(* CoDeSys 2.3.9.50 project: flat-BC9000.pr6 *)
(* Libraries: PlcHelperBC.lb6 7.5.01 11:03:00, COMlibV2.lb6 25.2.14 08:37:08, ModbusRTU.lb6 13.5.15 12:37:26, standard.lb6 5.6.98 11:03:02 *)

(* Global variable list: Globale_Variablen *)
VAR_GLOBAL

	Clear						: ClearComBuffer;
	TxBufferCom1				: ComBuffer;
	RxBufferCom1				: ComBuffer;
	SerialLineControlCom1			: SerialLineControl;
	ReceiveDataCom1			: ReceiveData;
	SendDataCom1				: SendData;

	Modbus						: Modbus_Struct;
	Internal						: Internal_Struct;

	HW_vent_out_level					AT	%QW2:WORD:=7000;(* Напряжение управления вытяжным вентилятором (0-32767) *)
(*	HW_vent_out_level2					AT	%QW6:WORD:=7000;
	HW_vent_out_level3					AT	%QW10:WORD:=7000;
	HW_vent_out_level4					AT	%QW14:WORD:=7000;
*)

(*	RS485read.MB.InData AT %IB16 : MB_KL6inData22B;
	RS485read.MB.OutData AT %QB16 : MB_KL6outData22B;
*)


	HW_temp_kitchen_box					AT %IW42:INT; (*Температура на кухне в коробе  *)
	HW_temp_vent_in						AT %IW46:INT; (*Температура притока перед фильтром *)
	HW_temp_street						AT %IW50:INT; (*Температура на улице *)
	HW_temp_bedroom					AT %IW54:INT; (*Температура в спальне *)

	HW_temp_child_small_room			AT %IW58:INT; (*Температура *)
	HW_temp_kitchen						AT %IW62:INT; (*Температура *)
	HW_temp_child_big_room				AT %IW66:INT; (*Температура *)


	HW_vent_in_trans_105_130				AT	%QX72.0:BOOL:=FALSE;  (* Напряжение 110 или 130 В *)
	HW_vent_in_trans_160_220				AT	%QX72.1:BOOL:=TRUE;  (* Напряжение 160 или 220 В *)
	HW_vent_in_trans_LO_HI				AT	%QX72.2:BOOL:=FALSE;  (* Напряжение 110/130  или 160/220 В *)
	HW_steam							AT	%QX72.3:BOOL:=FALSE; (* Разрешение включения увлажнителя *)

	HW_vent_out							AT	%QX72.4:BOOL:=FALSE; (* Вытяжной вентилятор*)
	HW_kitchen_vent_out					AT	%QX72.5:BOOL:=FALSE; (*Надплитная вытяжка*)
	HW_vent_in_heat_level				AT	%QX72.6:BOOL:=FALSE; (* Подогрев притока ночной режим   -5 К ТЭН *)
	HW_vent_valve						AT	%QX72.7:BOOL:=FALSE; (*Клапан приточной вентиляции"*)


	HW_valve_water_kitchen				AT	%QX73.0:BOOL; (* Кран ХВС и ГВС на кухне *)
	HW_valve_water_bathroom				AT	%QX73.1:BOOL; (* Кран ХВС и ГВС в санузле *)
	HW_LIGHT_ALL						AT	%QX73.2:BOOL; (*Свет в квартире *)
	HW_LIGHT_hall						AT	%QX73.3:BOOL; (*Ночной/аварийный свет в коридоре *)

(*
	HW_rez1								AT	%QX69.4:BOOL; 
	HW_rez2								AT	%QX69.5:BOOL; 
	HW_rez3								AT	%QX69.6:BOOL; 
	HW_rez4								AT	%QX69.7:BOOL;

*)

	HW_trans_power						AT	%QX74.0:BOOL:=FALSE; (*Подача тока на трансформатор и реле ТЭН-а *)
	HW_vent_in_heat						AT	%QX74.1:BOOL:=FALSE; (* Подогрев притока - ТЭН *)





	HW_sensor_fld_kitchen				AT %IX72.0:BOOL; (* Датчик протечки на кухне*)
	HW_sensor_fld_tlt						AT %IX72.1:BOOL; (* Датчик протечки в туалете*)
	HW_sensor_fld_post					AT %IX72.2:BOOL; (* Датчик протечки в постирочной*)
	HW_sensor_fld_van					AT %IX72.3:BOOL; (* Датчик протечки в ванной*)
	HW_impulse_kitchen_water_cold		AT %IX72.4:BOOL; (* Счётчик холодной воды на кухне*)
	HW_impulse_kitchen_water_warm		AT %IX72.5:BOOL; (* Счётчик горячей воды на кухне*)
	HW_vent_reay_pressure				AT %IX72.6:BOOL; (*Реле давления*)
	HW_kitchen_button_vent_out			AT %IX72.7:BOOL; (* Кнопка кухонной вытяжки*)

	HW_sensor_vent_valve_closed			AT %IX73.0:BOOL;
	HW_sensor_vent_valve_opened		AT %IX73.1:BOOL;
	HW_IN01							AT %IX73.2:BOOL;(*Кнопка вкл и откл света в квартире*)
	HW_IN02							AT %IX73.3:BOOL;(*Кнопка вкл и откл кранов воды на кухне*)
	HW_IN03							AT %IX73.4:BOOL;(*Кнопка вкл и откл кранов воды на кухне*)
	HW_IN04							AT %IX73.5:BOOL;(*Кнопка вкл и откл Вентиляции*)
	HW_IN05							AT %IX73.6:BOOL;(*Кнопка вкл и откл Резерв*)
	HW_gerkon							AT %IX73.7:BOOL;(*Датчик открытия двери - геркон*)


	HW_PIR_door						AT %IX74.0:BOOL;(*Датчик открытия двери - pir *)
	HW_PIR_hall							AT %IX74.1:BOOL;(*Датчик открытия двери - pir *)
	HW_electro							AT %IX74.2:BOOL;(*Датчик наличия электроэнергии*)
	HW_battery_low						AT %IX74.3:BOOL;(*Датчик низкого напряжения  АКБ*)



	HW_impulse_bathroom_water_cold		AT %IX75.0:BOOL; (* Счётчик горячей воды санузла NAMUR*)
	HW_impulse_bathroom_water_warm		AT %IX75.2:BOOL; (* Счётчик холодной воды санузла NAMUR*)







END_VAR

(* Global variable list: Variable_Configuration *)
VAR_CONFIG
	RS485read.MB.InData AT %IB16 : MB_KL6inData22B;
	RS485read.MB.OutData AT %QB16 : MB_KL6outData22B;
END_VAR

(* Data type *)
TYPE Internal_struct :
STRUCT

	Temp_vent_in						:	REAL; 		(*16434*)
	City_hum 							:	REAL;		(*16436*)
	Kitchen_room_tempout					:	REAL;		(*16438 *)

	Kitchen_room_temp 					:	REAL; 		(*16440 *)
	Kitchen_room_temp_SHT20 			:	REAL;		(*16442 *)
	Kitchen_room_hum 					:	REAL;		(*16444 *)
	Kitchen_room_CO2					:	REAL;		(*16446  *)

	Child_small_room_temp 				:	REAL; 		(* 16448 *)
	Child_small_room_temp_SHT20 		:	REAL;	(*16450 *)
	Child_small_room_hum 				:	REAL;	(*16452 *)
	Child_small_room_CO2 				:	REAL;	(* 16454 *)

	Child_big_room_temp	 				:	REAL; 	(* 16456 *)
	Child_big_room_temp_SHT20	 		:	REAL;	(* 16458 *)
	Child_big_room_hum	 				:	REAL;	(* 16460 *)
	Child_big_room_CO2	 				:	REAL;	(* 16462 *)

	Bed_room_temp	 					:	REAL; 	(* 16464 *)
	Bed_room_temp_SHT20				:	REAL;	(* 16466 *)
	Bed_room_hum	 					:	REAL;	(* 16468 *)
	Bed_room_CO2						:	REAL;	(*16470 *)

END_STRUCT
END_TYPE

(* Data type *)
TYPE Modbus_struct :
STRUCT

	(* MEED TO SAVE IN MEMORY*)



	Vent							AT %MB0	:	BOOL;	(*16384*)
	Vent_out						AT %MB2	:	BOOL;	(*16385*)
	Vent_heat					AT %MB4	:	INT;		(*16386*)
	Vent_heat_level				AT %MB6	:	BOOL;	(*16387*)
	Vent_valve_status				AT %MB8	:	INT;     	(*16388*)
	Steam						AT %MB10	:	BOOL;	(*16389*)
	Target_CO2					AT %MB12	:	INT;		(*16390*)
	Target_hum					AT %MB14	:	INT; 	(*16391*)
	Security_status				AT %MB16	:	BOOL;	(*16392*)
(*	Light_reserv					AT %MB18	:	BOOL;*)   (*16393*)
	Light						AT %MB20	:	BOOL; 	(*16394 *)
	Light_hall					AT %MB22	:	BOOL; 	(*16395*)

	Kitchen_stat_cold_water		AT %MD24	:	DINT; (* 16396*)
	Kitchen_stat_warm_water		AT %MD28	:	DINT; (* 16398*)
	Bathroom_stat_cold_water		AT %MD32	:	DINT; (* 16400*)
	Bathroom_stat_warm_water		AT %MD36	:	DINT; (* 16402*)

	FLD_valve_kitchen 			AT %MB40	:	BOOL; (* Положение  крана воды на кухне 16404*)
	FLD_valve_bathroom 			AT %MB42	:	BOOL; (*Положение  крана воды в санузле 16405*)
	FLD_ALRM_KITCHEN 			AT %MB44	:	BOOL; (*ТРЕВОГА ЗАТОПЛЕНИЕ НА КУХНЕ 16406*)
	FLD_ALRM_BATH 			AT %MB46	:	BOOL; (*ТРЕВОГА ЗАТОПЛЕНИЕ В САНУЗЛЕ 16407*)

	(* NOT NEED TO SAVE in MEMORY *)

	Steam_level						AT %MB48	:	INT;     (* 16408*)
	Steam_status						AT %MB50	:	INT;  (* 16409*)
	Steam_real						AT %MB52	:	INT; (* 16410*)
	Vent_input_level					AT %MB54	:	INT;		(*16411*)
	Vent_output_level					AT %MB56	:	INT; 	(*0-100%    16412 *)
	Vent_pressure_relay				AT %MB58	:	BOOL; (* 16413*)


	Gerkon							AT %MB60	:	BOOL; (*Датчик открытия входной двери (геркон)    16414 *)
	PIR_door						AT %MB62	:	BOOL;(*Датчик открытия входной двери PIR-штора   16415 *)
	Power_supply					AT %MB64	:	BOOL;(*Электроэнергия   16416 *)
	Battery_low						AT %MB66	:	BOOL;	(* 16417*)
	Rezerv							AT %MB68	:	BOOL; (* 16418*)

	FLD_PRC						AT %MB70	:	BOOL; (*Датчик в постирочной 16419*)
	FLD_TLT						AT %MB72	:	BOOL; (*Датчик в туалете 16420*)
	FLD_BATH						AT %MB74	:	BOOL;(*Датчик в  ванной 16421*)
	FLD_KUH						AT %MB76	:	BOOL;(*Датчик на  кухне 16422*)

	Uv								AT %MW80	:	DINT;		(*16424*)
	Ia								AT %MW84	:	DINT;		(*16426*)
	Pw								AT %MW88	:	DINT;		(*16428*)
	E_T1							AT %MW92	:	DINT;		(*16430*)
	E_T2							AT %MW96	:	DINT;		(*16432*)


	Temp_vent_in					AT %MW100	:	DINT; 		(*16434*)
	City_hum 						AT %MW104	:	DINT;		(*16436*)
	Kitchen_room_tempout				AT %MW108	:	DINT;		(*16438 *)

	Kitchen_room_temp 				AT %MW112	:	DINT; 		(*16440 *)
	Kitchen_room_temp_SHT20 		AT %MW116	:	DINT;		(*16442 *)
	Kitchen_room_hum 				AT %MW120	:	DINT;		(*16444 *)
	Kitchen_room_CO2				AT %MW124	:	DINT;		(*16446  *)

	Child_small_room_temp 			AT %MW128	:	DINT; 		(* 16448 *)
	Child_small_room_temp_SHT20 	AT %MW132	:	DINT;	(*16450 *)
	Child_small_room_hum 			AT %MW136	:	DINT;	(*16452 *)
	Child_small_room_CO2 			AT %MW140	:	DINT;	(* 16454 *)

	Child_big_room_temp	 			AT %MW144	:	DINT; 	(* 16456 *)
	Child_big_room_temp_SHT20	 	AT %MW148	:	DINT;	(* 16458 *)
	Child_big_room_hum	 			AT %MW152	:	DINT;	(* 16460 *)
	Child_big_room_CO2	 			AT %MW156	:	DINT;	(* 16462 *)

	Bed_room_temp	 				AT %MW160	:	DINT; 	(* 16464 *)
	Bed_room_temp_SHT20			AT %MW164	:	DINT;	(* 16466 *)
	Bed_room_hum	 				AT %MW168	:	DINT;	(* 16468 *)
	Bed_room_CO2					AT %MW172	:	DINT;	(*16470 *)





END_STRUCT
END_TYPE

(* POU MAIN, ST *)
PROGRAM MAIN
VAR
	SW_LIGHT				: SM_BUTT;		(* вкл/откл  света в квартире *)
	SW_VALVE_BATH		: SM_BUTT;
	SW_VALVE_KITCHEN		: SM_BUTT;
	SW_VENT				: SM_BUTT_SHORT_LONG;		(* вкл/откл вентиляции *)
	SW_REZERV			: SM_BUTT_TIMER;

END_VAR
	RS485read;				(* Работа с устройствами на шине RS485 *)
	Ventcontrol;				(* Глобальный контроль вентустановки*)
	VentPower;				(* Авторегулировка мощности вентустановки по датчикам CO2*)
	Counters;				(* Счётчики воды *)
	Fluid_bath;				(* Защита от протечки в санузлах. Оработка нажатия физической и виртульной кнопки №2 *)
	Fluid_kitchen;				(* Защита от протечки в кухне. Оработка нажатия физической и виртульной кнопки №3 *)
	Light_hall;				(* Свет в коридоре *)




(* Оработка нажатия физических и виртульных кнопок №1, №4, №5 *)

	SW_LIGHT 				(IN:=HW_IN01, IN1:= Modbus.Light, 	Q=>NOT Modbus.Light);	(* Конпка №1 *)
	SW_VALVE_BATH 		(IN:=HW_IN02, IN1:= Modbus.FLD_valve_bathroom, 	Q=>NOT Modbus.FLD_valve_bathroom);	(* Конпка №2 *)
	SW_VALVE_KITCHEN 	(IN:=HW_IN03, IN1:= Modbus.FLD_valve_kitchen,	Q=>NOT Modbus.FLD_valve_kitchen);	(* Конпка №3 *)
	SW_VENT 				(bIn:=HW_IN04, TC:=t#2000ms);		(* Конпка №4  , обработка короткого и долгого нажатия *)
	SW_REZERV		 	(IN:=HW_IN05,Q=>);	(* Конпка №3 *)

	IF	SW_VENT.bSingle	THEN
		Modbus.Vent	:= NOT Modbus.Vent;
	END_IF

	IF	SW_VENT.bLong	THEN
		Modbus.Steam	:= NOT Modbus.Steam;
	END_IF

(* Прямая связь между экспортирумымми переменными и  переменными, жестко привязаными  к физ. портам. Частота обновления= циклу ПЛК  : *)

	HW_LIGHT_ALL				:=	NOT Modbus.Light;				(* СВЕТ в квартире*)
	HW_LIGHT_HALL				:=	Modbus.Light_hall;					(* Аварийный СВЕТ в квартире*)
	Modbus.Gerkon				:=	HW_gerkon;						(* Геркон на двери*)
	Modbus.PIR_door				:=	HW_pir_door;						(* Датчик движения на двери *)
	Modbus.Power_supply			:=	HW_electro;						(* Датчик наличия электроэнергии *)
	Modbus.Battery_low			:=	HW_battery_low;					(* Датчик наличия электроэнергии *)
	Modbus.Vent_pressure_relay	:=	HW_vent_reay_pressure; 	(* Relay pressure *)
	HW_vent_in_heat_level		:=	Modbus.Vent_heat_level;

	Internal.Temp_vent_in				:=	INT_TO_REAL(HW_temp_vent_in)/10;
	Internal.Kitchen_room_tempout		:=	INT_TO_REAL(HW_temp_street)/10;
	Internal.Bed_room_temp			:=	INT_TO_REAL(HW_temp_bedroom)/10;
	Internal.Kitchen_room_temp			:=	INT_TO_REAL(HW_temp_kitchen)/10;
	Internal.Child_big_room_temp		:=	INT_TO_REAL(HW_temp_child_big_room)/10;
	Internal.Child_small_room_temp		:=	INT_TO_REAL(HW_temp_child_small_room)/10;



	Modbus.Temp_vent_in				:=	INT_TO_DINT(HW_temp_vent_in);
	Modbus.Kitchen_room_tempout		:=	INT_TO_DINT(HW_temp_street);
	Modbus.Bed_room_temp			:=	INT_TO_DINT(HW_temp_bedroom);
	Modbus.Kitchen_room_temp		:=	INT_TO_DINT(HW_temp_kitchen);
	Modbus.Child_big_room_temp		:=	INT_TO_DINT(HW_temp_child_big_room);
	Modbus.Child_small_room_temp	:=	INT_TO_DINT(HW_temp_child_small_room);


IF (Modbus.Security_status = FALSE AND HW_electro = FALSE  ) THEN
	Modbus.Light_hall :=TRUE;
END_IF

IF (Modbus.Security_status = TRUE ) THEN
	Modbus.Light_hall := FALSE;
END_IF
END_PROGRAM

(* POU SM_BUTT, ST *)
FUNCTION_BLOCK SM_BUTT            (* ФУНКЦИОНАЛЬНЫЙ БЛОК ДЛЯ ПРОСТОЙ КНОПКИ *)
    VAR_INPUT
       	IN: BOOL;          	(*ВХОД ЗА КОТОРЫМ МЫ СЛЕДИМ *)
	IN1:BOOL;				(*ВЫХОД ЗА КОТОРЫМ ТОЖЕ СЛЕДИМ*)
    END_VAR

    VAR_OUTPUT
	Q : BOOL;        			(*СОСТОЯНИЕ ВЫХОДА*)
    END_VAR
    VAR
  MEM : BOOL;    			(* ВНУТРЕННЯЯ ПЕРЕМЕННАЯ ДЛЯ ХРАНЕНИЯ СОСТОЯНИЯ КНОПКИ *)
    END_VAR
Q:=IN1;

IF IN AND NOT MEM THEN 	(* ПОЙМАЛИ ПЕРЕДНИЙ ФРОНТ - НАЖАЛИ НА КНОПКУ *)
	Q := NOT IN1;    			(* МЕНЯЕМ СОСТОЯНИЕ ВЫХОДА НА ПРОТИВОПОЛОЖНОЕ *)
END_IF

MEM := IN;                       		(* ЗАПОМИНАЕМ ТЕКУЩЕЕ ЗНАЧЕНИЕ КНОПКИ *)
END_FUNCTION_BLOCK

(* POU SM_BUTT_SHORT_LONG, ST *)
FUNCTION_BLOCK SM_BUTT_SHORT_LONG
VAR_INPUT
	bIn 	: BOOL;
	TC	: TIME := t#2000ms;
END_VAR
VAR_OUTPUT
	bSingle	: BOOL;
	bLong 	: BOOL;
END_VAR
VAR
	timer 	: TP;
	ft1		: F_TRIG;
	ft2		: F_TRIG;
END_VAR
timer(in := bIn, pt := TC);

ft1(clk := bIn);
bSingle := ft1.Q AND timer.Q;

ft2(clk := timer.Q);
bLong := ft2.Q AND bIn;
END_FUNCTION_BLOCK

(* POU SM_BUTT_TIMER, ST *)
FUNCTION_BLOCK SM_BUTT_TIMER            (* ФУНКЦИОНАЛЬНЫЙ БЛОК ДЛЯ ПРОСТОЙ КНОПКИ *)
    VAR_INPUT
       	IN: BOOL;          	(*ВХОД ЗА КОТОРЫМ МЫ СЛЕДИМ *)
    END_VAR

    VAR_OUTPUT
	Q : BOOL;        			(*СОСТОЯНИЕ ВЫХОДА*)
    END_VAR

VAR
	RT1				: R_TRIG;
	tmCheck			: TON;
END_VAR
tmCheck;

RT1(clk := IN);

IF RT1.Q THEN
	Modbus.Rezerv	:=	TRUE;
	tmCheck(in:=FALSE);
	tmCheck(in:=TRUE,pt:=t#2s);
END_IF

IF tmCheck.Q	THEN
		Modbus.Rezerv	:=	FALSE;
END_IF
END_FUNCTION_BLOCK

(* POU RS485read, ST *)
PROGRAM RS485read
VAR
	MB: ModbusRtuMaster_KL6x22B;
	timeoutvalue					: TIME := T#500ms;		(* timeout while waiting for an answer of the modbus slave *)
	delta_sensor_hum				: INT:=10;					(*Корректировка показаний датчика, % относительной влажности*)
	Period_steam				: INT := 60; 				(* Частота изменения уставки мощности  увлажнителя, секунды*)
	Period_modbus				: INT := 10;  				(* Частота опроса устройств modbus, секунды*)

	r_Target_hum					: REAL;
	r_room_hum					: REAL;
	i_Steam_level				: INT:=0;
	MBdata						: ARRAY [1..2] OF INT;		(* The size of this array can be adapted to the modbus slaves register area *)

	sensors_SHT20_v1_id			: ARRAY[1..4] OF BYTE:=16#01, 16#02, 16#03, 16#37;
	sensors_SHT20_v1_hum		: ARRAY[1..4] OF REAL:=4(0);
	sensors_SHT20_v1_temp		: ARRAY[1..4] OF REAL:=4(0);


	sensors_CO2_id				: ARRAY[1..4] OF BYTE:=16#68, 16#65, 16#66, 16#67;
	sensors_CO2_ppm			: ARRAY[1..4] OF REAL;

	FtrigBusy					: F_TRIG;
	state						: INT;
	busy						: BOOL;
	LastErrorstate					: INT;
	LastModbusError				: ST_ModbusErrorDiagnostics;
	CounterError					: DINT;
	CounterSuccess				: DINT;
	tmCheck						: TON;
	Timer1						: TON;
	Timer2						: TON;
	Timer1Q						: BOOL;
	Timer2Q						: BOOL;
	Hum_old						: REAL;
	Steam_response				: WORD:=0;
	tTimerValue					: TIME;
	tTimerValue_modbus			: TIME;
	get_run_Merc200_done		: BOOL;
	get_hist_Merc200_done		: BOOL;
	get_run_Merc200				: FB_GET_RUN_MERC200;
	get_hist_Merc200				: FB_GET_HIST_MERC200;


	i: INT:=1;
	k: INT:=1;

END_VAR
tmcheck();
Timer1();
Timer2();

CASE state OF

0:
		MB.ReadRegs(Execute:= FALSE);
		state := 2;


 2:
	Clear(Buffer := RxBufferCom1);


		MB.ReadRegs(
			UnitID:= sensors_SHT20_v1_id[i],
			Quantity:= 2,
			MBAddr:= 0,
			cbLength:= 6,
			pMemoryAddr:= ADR(MBdata),
			Execute:= TRUE,
			Timeout:= timeoutvalue,
			Busy => busy,
		);
		IF NOT busy THEN
			IF (mb.Error = FALSE ) THEN
				sensors_SHT20_v1_temp[i]:=INT_TO_REAL(MBdata[1]);
				sensors_SHT20_v1_hum[i]:=INT_TO_REAL(MBdata[2])- 10*delta_sensor_hum;
			END_IF
			i:=i+1;
			MB.ReadRegs(Execute:= FALSE);
			IF (i>4 )	THEN
				i:=1;

				Internal.Kitchen_room_hum				:=	sensors_SHT20_v1_hum[1];
				Internal.Bed_room_hum				:=	sensors_SHT20_v1_hum[2];
				Internal.Child_big_room_hum			:=	sensors_SHT20_v1_hum[3];
				Internal.Child_small_room_hum			:=	sensors_SHT20_v1_hum[4];

(*				Internal.Kitchen_room_temp_SHT20		:=	sensors_SHT20_v1_temp[1];
				Internal.Bed_room_temp_SHT20			:=	sensors_SHT20_v1_temp[2];
				Internal.Child_small_room_temp_SHT20	:=	sensors_SHT20_v1_temp[4];
				Internal.Child_big_room_temp_SHT20	:=	sensors_SHT20_v1_temp[3];

				Modbus.Kitchen_room_temp_SHT20		:=	REAL_TO_INT(sensors_SHT20_v1_temp[1]);
				Modbus.Bed_room_temp_SHT20		:=	REAL_TO_INT(sensors_SHT20_v1_temp[2]);
				Modbus.Child_big_room_temp_SHT20	:=	REAL_TO_INT(sensors_SHT20_v1_temp[3]);
				Modbus.Child_small_room_temp_SHT20	:=	REAL_TO_INT(sensors_SHT20_v1_temp[4]);
*)
				Modbus.Kitchen_room_hum				:=	REAL_TO_INT(sensors_SHT20_v1_hum[1]);
				Modbus.Bed_room_hum				:=	REAL_TO_INT(sensors_SHT20_v1_hum[2]);
				Modbus.Child_big_room_hum			:=	REAL_TO_INT(sensors_SHT20_v1_hum[3]);
				Modbus.Child_small_room_hum			:=	REAL_TO_INT(sensors_SHT20_v1_hum[4]);
				state :=26;
			ELSE
				state :=2;
			END_IF

		END_IF


26:
		MB.ReadInputRegs(
			UnitID:=sensors_CO2_id[k], (* station address *)
			Quantity:= 1,
			MBAddr:= 3,
			cbLength:= 4,
			pMemoryAddr:= ADR(MBdata),
			Execute:= TRUE,
			Timeout:= timeoutvalue,
			Busy => busy	);
		IF NOT busy THEN
			IF (mb.Error = FALSE ) THEN
				sensors_CO2_ppm[k]	:=	INT_TO_REAL(MBdata[1]);
			END_IF
			k:=k+1;
			MB.ReadRegs(Execute:= FALSE);
			IF (k>4 )	THEN
				k:=1;
				Internal.Kitchen_room_CO2		:=	sensors_CO2_ppm[1];
				Internal.Bed_room_CO2		:=	sensors_CO2_ppm[2];
				Internal.Child_big_room_CO2	:=	sensors_CO2_ppm[3];
				Internal.Child_small_room_CO2	:=	sensors_CO2_ppm[4];

				Modbus.Kitchen_room_CO2		:=	REAL_TO_DINT(sensors_CO2_ppm[1]);
				Modbus.Bed_room_CO2		:=	REAL_TO_DINT(sensors_CO2_ppm[2]);
				Modbus.Child_big_room_CO2	:=	REAL_TO_DINT(sensors_CO2_ppm[3]);
				Modbus.Child_small_room_CO2	:=	REAL_TO_DINT(sensors_CO2_ppm[4]);

				state :=47;
			ELSE
				state :=26;
			END_IF
		END_IF

47:	(*Изменение уставки мощности увлажнителя при необходимости с частотой Period_steam *)

		IF (Modbus.Steam=TRUE AND Modbus.Vent=TRUE ) THEN
			r_Target_hum:=INT_TO_REAL( Modbus.Target_Hum) ;
			r_room_hum:=DINT_TO_REAL(Modbus.Bed_room_hum)/10;
			tTimerValue := t#60s;
			Timer2(IN:=NOT Timer2Q , PT:=tTimerValue , Q=>Timer2Q , ET=> );
			IF timer2.q THEN
				IF  ( r_room_hum <= r_Target_hum*0.5 AND i_Steam_level< 50 ) THEN
					i_Steam_level:=50;
				END_IF

				IF ( ( r_room_hum <=   Hum_old )
				AND ( r_room_hum > r_Target_hum*0.5)
				AND ( r_room_hum < r_Target_hum*0.95 )) THEN
					i_Steam_level:=i_Steam_level+1;
				END_IF

				IF ( r_room_hum >= r_Target_hum*1.05) THEN
					i_Steam_level:=i_Steam_level-1;
				END_IF

				Hum_old:=r_room_hum;

			END_IF

			IF (i_Steam_level>100) THEN
				i_Steam_level:=100;
			END_IF

			IF (i_Steam_level<10) THEN
				i_Steam_level:=10;
			END_IF

			Modbus.Steam_level:=INT_TO_BYTE(i_Steam_level);

			MB.WriteSingleRegister(
					UnitID:= 16#0A, (* station address *)
					Quantity:= 1,
					MBAddr:= 1537,
					cbLength:= 2,
					pMemoryAddr:= ADR(Modbus.Steam_level),
					Execute:= TRUE,
					Timeout:= timeoutvalue,
					Busy => busy	);
			IF NOT busy THEN
					MB.WriteSingleRegister(Execute:= FALSE);
					state := 77;
			END_IF
		ELSE
			Modbus.Steam_level:=0;
			state := 77;
		END_IF


77:		(* Фактический процент текущей  мощности увлажнителя *)

			MB.ReadRegs(
					UnitID:= 16#0A, (* station address *)
					Quantity:= 1,
					MBAddr:= 261,
					cbLength:= 2,
					pMemoryAddr:= ADR(Steam_response),
					Execute:= TRUE,
					Timeout:= timeoutvalue,
					Busy => busy	);
				IF NOT busy THEN
					IF (mb.Error = FALSE ) THEN
						Modbus.Steam_real:=Steam_response;
					END_IF
					MB.ReadRegs(Execute:= FALSE);
					state := 79;

				END_IF


79:
		tmCheck(in:=FALSE);
		tmCheck(in:=TRUE,pt:=t#2s);
		get_run_Merc200_done := FALSE;
		busy:=TRUE;
		get_run_Merc200( Uv=>Modbus.Uv,Ia=>Modbus.Ia,Pw=>Modbus.Pw, done=>get_run_Merc200_done);
		IF get_run_Merc200_done = TRUE THEN

			busy:=FALSE;
			state:=80;
		ELSIF tmcheck.Q THEN
			busy:=FALSE;
			 state:=80;
		END_IF

80:
		tmCheck(in:=FALSE);
		tmCheck(in:=TRUE,pt:=t#2s);
		get_hist_Merc200_done := FALSE;
		busy:=TRUE;
		get_hist_Merc200( E_T1=>Modbus.E_T1,E_T2=>Modbus.E_T2, done=>get_hist_Merc200_done);
		IF get_hist_Merc200_done = TRUE THEN

			busy:=FALSE;
			state:=88;
		ELSIF tmcheck.Q THEN
			busy:=FALSE;
			 state:=88;
		END_IF

88:
		tTimerValue_modbus := t#10s;
		Timer1(IN:=NOT Timer1Q , PT:=tTimerValue_modbus , Q=>Timer1Q , ET=> );
		IF timer1.q THEN

			state:=0;
		END_IF

END_CASE

FtrigBusy(CLK:=mb.BUSY );
IF FtrigBusy.Q THEN
	IF mb.Error THEN
		LastModbusError := mb.ErrorDiagnostics;
		LastErrorstate := state;
		CounterError := CounterError + 1;
	ELSE
		CounterSuccess := CounterSuccess + 1;
	END_IF
END_IF

SerialLinecontrolCom1(
	mode:=SerialLinemode_kl6_22b_standard,
	pComIn:=ADR(RS485read.MB.InData),
	pComOut:=ADR(RS485read.MB.OutData),
	SizeComIn:=SIZEOF(RS485read.MB.OutData),
	TxBuffer:=TxBufferCom1,
	RxBuffer:=RxBufferCom1,
	Error=>,
	errorid=>);
END_PROGRAM

(* POU FB_GET_RUN_MERC200, ST *)
FUNCTION_BLOCK FB_GET_RUN_MERC200
VAR_INPUT

END_VAR

VAR_OUTPUT
	Uv				: DINT;
	Ia				: DINT;
	Pw				: DINT;
	done			: BOOL;
END_VAR

VAR
	SendBuffer		: ARRAY[1..7] OF BYTE;
	ReceiveBuffer	: ARRAY[1..14] OF BYTE;
	Clear			: ClearComBuffer;
	state			: INT:= 0;
	tmcheck			: TON;

	crctest			: WORD;
	Uv_word			: WORD;
	Ia_word			: WORD;
	Pw_dword		: DWORD;

	CRC_calc: WORD;
	CRC_get: WORD := 1;

END_VAR
tmcheck();

CASE state OF

0:
	done:=FALSE;
	Clear(Buffer := RxBufferCom1);
	SendBuffer[1] := 16#00;

	SendBuffer[2] := 16#0B; (* Address  dec 740964 = hex 0B 4E 64  *)
	SendBuffer[3] := 16#4E; (* Address *)
	SendBuffer[4] := 16#64; (* Address *)

	SendBuffer[5] := 16#63; (*Command*)
	crctest:=F_CRC16(ADR(SendBuffer), 5);
	MEMCPY(ADR(SendBuffer)+5,ADR(crctest),2);

	SendDataCom1(pSendData:=ADR(SendBuffer),length:=7,TXbuffer:=TXBufferCom1,Busy=>,Error=>);

	tmCheck(in:=FALSE);
	tmCheck(in:=TRUE,pt:=t#2s);
	state:=1;

1: (*ответ*)

	ReceiveDataCom1(pPrefix:=,LenPrefix:=,pSuffix:=,LenSuffix:=,pReceiveData:=ADR(ReceiveBuffer),SizeReceiveData:=14,TImeOut:=t#2s,Reset:=,RXbuffer:=RxBufferCom1,DataReceived=>,busy=>,RxTimeout=>,LenReceiveData=>);

	IF ReceiveDataCom1.Error <> 0 THEN
		state:=9;
	END_IF

	IF ReceiveDataCom1.DataReceived THEN
		state:=2;
	ELSIF tmcheck.Q THEN
		 state:=9;
	END_IF;



2:(*расшифровка*)
	CRC_calc := F_CRC16(ADR(ReceiveBuffer), 12);
	MEMCPY(ADR(CRC_get),ADR(ReceiveBuffer[13]),1);
	MEMCPY(ADR(CRC_get)+1,ADR(ReceiveBuffer[14]),1);


	IF (  ReceiveBuffer[1] = 16#00  AND CRC_calc = CRC_get ) THEN

		MEMCPY(ADR(Uv_word),ADR(ReceiveBuffer[7]),1);
		MEMCPY(ADR(Uv_word)+1,ADR(ReceiveBuffer[6]),1);
		Uv:=STRING_TO_DINT(DWORD_TO_STRH(Uv_word));



		MEMCPY(ADR(Ia_word),ADR(ReceiveBuffer[9]),1);
		MEMCPY(ADR(Ia_word)+1,ADR(ReceiveBuffer[8]),1);
		Ia:=STRING_TO_DINT(DWORD_TO_STRH(Ia_word));

		MEMCPY(ADR(Pw_dword),ADR(ReceiveBuffer[12]),1);
		MEMCPY(ADR(Pw_dword)+1,ADR(ReceiveBuffer[11]),1);
		MEMCPY(ADR(Pw_dword)+2,ADR(ReceiveBuffer[10]),1);
		Pw:=STRING_TO_DINT(DWORD_TO_STRH(Pw_dword));


		state:=10;
	ELSE
		state:=9;
	END_IF

9:
	Uv:=0;
	done := TRUE;
	state:=0;
10:
	done := TRUE;
	state:=0;

END_CASE;
END_FUNCTION_BLOCK

(* POU MB_func/F_CRC16, ST *)
FUNCTION F_CRC16 : WORD
VAR_INPUT
	pData: POINTER TO BYTE;		(* указатель на блок данных *)
	Size: WORD;						(* размер блока  данных *)
END_VAR
VAR
	Cnt: BYTE;							(* счетчик битов *)
END_VAR
F_CRC16 := 16#FFFF;
WHILE Size > 0 DO
	F_CRC16 := F_CRC16 XOR pData^;
	FOR Cnt := 0 TO 7 DO
		IF F_CRC16.0 = 0 THEN
			F_CRC16 := SHR(F_CRC16, 1);
		ELSE
			F_CRC16 := SHR(F_CRC16, 1) XOR 16#A001;
		END_IF
	END_FOR;
	pData := pData + 1;
	Size := Size - 1;
END_WHILE
END_FUNCTION

(* POU DWORD_TO_STRH, ST *)
FUNCTION DWORD_TO_STRH : STRING(8)
VAR_INPUT
	IN : DWORD;
END_VAR
VAR
	i : INT;
	temp : BYTE;
	pt : POINTER TO BYTE;
END_VAR
(*
version 1.3	29. mar. 2008
programmer 	hugo
tested by	tobias

DWORD_TO_STRINGH converts a DWORD to a String of Hexadecimal represented by '0' .. '9' and 'A' .. 'F'.
The lowest order Character will be on the right and the high order Character on the left.

*)

(* @END_DECLARATION := '0' *)
(* read output adress to pointer *)
pt := ADR(DWORD_TO_STRH) + 8;
(* wirte the closing byte for the string *)
pt^:= 0;

(* write the 8 hex characters backwards *)
FOR i := 1 TO 8 DO;
	(* decrement the pointer *)
	pt := pt - 1;
	(* read the lowest order hex value *)
	temp := DWORD_TO_BYTE(in AND 16#0000000F);
	(* convert value to hex character *)
	IF temp <= 9 THEN temp := temp + 48; ELSE temp := temp + 55; END_IF;
	(* write character to output string *)
	PT^ := temp;
	(* shift in for nect hex character *)
	in := SHR(in,4);
END_FOR;


(* code beofre rev 1.2
FOR i := 1 TO 8 DO
	X := DWORD_TO_BYTE(in AND 2#1111);
	IF X <= 9 THEN X := X + 48; ELSE X := X + 55; END_IF;
	Cx := CHR(X);
	temp := CONCAT(Cx, temp);
	in := SHR(in,4);
END_FOR;
DWORD_TO_STRH := temp;
*)


(* revision history
hm	9. jun. 2007	rev 1.0		
	original version 

hm	11. sep. 2007	rev 1.1
	changed coding for compatibility with twincat, concat cannot support a function as an argument.

hm	15. dec. 2007	rev 1.2
	changed code for better performance

hm	29. mar. 2008	rev 1.3
	changed STRING to STRING(8)

*)
END_FUNCTION

(* POU FB_GET_HIST_MERC200, ST *)
FUNCTION_BLOCK FB_GET_HIST_MERC200
VAR_INPUT

END_VAR

VAR_OUTPUT
	E_T1			: DINT;
	E_T2			: DINT;
(*	E_T3			: REAL;
	E_T4			: REAL;
*)
	done			: BOOL;
END_VAR

VAR
	SendBuffer		: ARRAY[1..7] OF BYTE;
	ReceiveBuffer	: ARRAY[1..23] OF BYTE:=0,0,0,0,0,0,0,0,0,0,0,0,0,0,0,0,0,0,0,0,0,0,0;
	Clear			: ClearComBuffer;
	state			: INT:= 0;
	tmcheck			: TON;

	crctest			: WORD;
	T1_dword		: DWORD;
	T2_dword		: DWORD;
(*	T3_dword		: DWORD;
	T4_dword		: DWORD;
*)
	CRC_calc: WORD;
	CRC_get: WORD := 1;

END_VAR
tmcheck();

CASE state OF

0:
	done:=FALSE;
	Clear(Buffer := RxBufferCom1);
	SendBuffer[1] := 16#00;

	SendBuffer[2] := 16#0B; (* Address  dec 740964 =0B 4E 64    *)
	SendBuffer[3] := 16#4E; (* Address *)
	SendBuffer[4] := 16#64; (* Address *)

	SendBuffer[5] := 16#27; (*Command*)

	crctest:=F_CRC16(ADR(SendBuffer), 5);
	MEMCPY(ADR(SendBuffer)+5,ADR(crctest),2);

	SendDataCom1(pSendData:=ADR(SendBuffer),length:=7,TXbuffer:=TXBufferCom1,Busy=>,Error=>);

	tmCheck(in:=FALSE);
	tmCheck(in:=TRUE,pt:=t#2s);
	state:=1;

1: (*ответ*)

	ReceiveDataCom1(pPrefix:=,LenPrefix:=,pSuffix:=,LenSuffix:=,pReceiveData:=ADR(ReceiveBuffer),SizeReceiveData:=23,TImeOut:=t#2s,Reset:=,RXbuffer:=RxBufferCom1,DataReceived=>,busy=>,RxTimeout=>,LenReceiveData=>);

	IF ReceiveDataCom1.Error <> 0 THEN
		state:=9;
	END_IF

	IF ReceiveDataCom1.DataReceived THEN
		state:=2;
	ELSIF tmcheck.Q THEN
		 state:=9;
	END_IF;



2:(*расшифровка*)
	CRC_calc := F_CRC16(ADR(ReceiveBuffer), 21);
	MEMCPY(ADR(CRC_get),ADR(ReceiveBuffer[22]),1);
	MEMCPY(ADR(CRC_get)+1,ADR(ReceiveBuffer[23]),1);


	IF (  ReceiveBuffer[1] = 16#00  AND ReceiveBuffer[2] = 16#0B AND ReceiveBuffer[3] = 16#4E AND ReceiveBuffer[4] = 16#64  AND ReceiveBuffer[5] = 16#27) THEN

		MEMCPY(ADR(T1_dword),ADR(ReceiveBuffer[9]),1);
		MEMCPY(ADR(T1_dword)+1,ADR(ReceiveBuffer[8]),1);
		MEMCPY(ADR(T1_dword)+2,ADR(ReceiveBuffer[7]),1);
		MEMCPY(ADR(T1_dword)+3,ADR(ReceiveBuffer[6]),1);
		E_T1:=STRING_TO_DINT(DWORD_TO_STRH(T1_dword));
(*		E_T1:=DWORD_TO_DINT(T1_dword); *)

		MEMCPY(ADR(T2_dword),ADR(ReceiveBuffer[13]),1);
		MEMCPY(ADR(T2_dword)+1,ADR(ReceiveBuffer[12]),1);
		MEMCPY(ADR(T2_dword)+2,ADR(ReceiveBuffer[11]),1);
		MEMCPY(ADR(T2_dword)+3,ADR(ReceiveBuffer[10]),1);
		E_T2:=STRING_TO_DINT(DWORD_TO_STRH(T2_dword));
(*		E_T2:=DWORD_TO_DINT(T2_dword); *)
(*
		MEMCPY(ADR(T3_dword),ADR(ReceiveBuffer[17]),1);
		MEMCPY(ADR(T3_dword)+1,ADR(ReceiveBuffer[16]),1);
		MEMCPY(ADR(T3_dword)+2,ADR(ReceiveBuffer[15]),1);
		MEMCPY(ADR(T3_dword)+3,ADR(ReceiveBuffer[14]),1);
		E_T3:=0.01*STRING_TO_REAL(DWORD_TO_HEXSTR(T3_dword,1,FALSE));

		MEMCPY(ADR(T4_dword),ADR(ReceiveBuffer[21]),1);
		MEMCPY(ADR(T4_dword)+1,ADR(ReceiveBuffer[20]),1);
		MEMCPY(ADR(T4_dword)+2,ADR(ReceiveBuffer[19]),1);
		MEMCPY(ADR(T4_dword)+3,ADR(ReceiveBuffer[18]),1);
		E_T4:=0.01*STRING_TO_REAL(DWORD_TO_HEXSTR(T4_dword,1,FALSE));
*)
		state:=10;
	ELSE
		state:=9;
	END_IF

9:
	E_T1:=0;
	E_T2:=0;

	done := TRUE;
	state:=0;
10:
	done := TRUE;
	state:=0;

END_CASE;
END_FUNCTION_BLOCK

(* POU Ventcontrol, ST *)
PROGRAM VentControl
VAR
	Temperature_max_to_heat		: REAL:=17;		(* Максимальная температура наружнего воздуха при которой разрешено включать воздухонагреватель *)
	Temperature_min_for_steam	: REAL:=14;		(* Минимальная температура воздуха в вент канале для разрешения работы увлажнителя *)
	gisterezis					: REAL:=0.2;		(* Гистерезис  разрешения включения воздухонагревателя, градусы цельсия *)


END_VAR
(* Состояние приточного клапана *)

IF (HW_sensor_vent_valve_opened=TRUE) THEN
	Modbus.Vent_valve_status:=1;
END_IF

IF (HW_sensor_vent_valve_closed=TRUE) THEN
	Modbus.Vent_valve_status:=0;
END_IF

IF (HW_sensor_vent_valve_closed=FALSE AND HW_sensor_vent_valve_opened=FALSE) THEN
	Modbus.Vent_valve_status:=2;
END_IF


IF (HW_kitchen_button_vent_out=TRUE) THEN	(* Если активирована кнопка надплитной вытяжки*)
	HW_vent_out:=TRUE;						(* Включаем вытяжной вент *)
	HW_vent_out_level:=32767;					(* Подаём управляющий сигнал DC на максимум *)
	HW_kitchen_vent_out:=TRUE;				(* Включаем вент надплитной вытяжки *)
ELSE
	HW_kitchen_vent_out:=FALSE;				(* Оключаем вент надплитной вытяжки *)
	IF (Modbus.Vent_out=FALSE) THEN			(* Если уставка работы вытяжного вента = FALSE*)
		HW_vent_out:=FALSE;					(* Отключаем вытяжной вент *)
	ELSE
		HW_vent_out:=TRUE;					(*  Включаем вытяжной вент  *)
	END_IF
END_IF


IF (Modbus.Vent=FALSE) THEN
	HW_steam:=FALSE;
	HW_vent_in_heat:=FALSE;
	HW_vent_valve:=FALSE; 	(* COMMENT THIS LINE TEMPORARY  ЛЕТНИЙ РЕЖИМ  !!!!!!!!!!!!!!!!!!!!!!!!!!!!!!!!!!!*)
	HW_trans_power:=FALSE;
ELSE
	HW_vent_valve:=TRUE;
	IF (HW_sensor_vent_valve_opened=TRUE) THEN
		HW_trans_power:=TRUE;
		IF (HW_vent_reay_pressure=TRUE) THEN

			IF (Modbus.Steam=TRUE)	THEN
				IF (Internal.Temp_vent_in>Temperature_min_for_steam+gisterezis) THEN
					HW_steam:=Modbus.Steam;
				END_IF
			IF (Internal.Temp_vent_in<Temperature_min_for_steam-gisterezis) THEN
					HW_steam:=Modbus.Steam;
				END_IF

			ELSE
				HW_steam:=FALSE;
			END_IF






			IF (Modbus.Vent_heat=2) THEN
				IF (Internal.Kitchen_room_tempout < Temperature_max_to_heat-gisterezis) THEN
					HW_vent_in_heat:=TRUE;
				(*	IF (Modbus.Vent_heat_level=TRUE) THEN
						HW_vent_in_heat_level:=TRUE;
					END_IF  *)
				END_IF
				IF (Internal.Kitchen_room_tempout > Temperature_max_to_heat+gisterezis) THEN
					HW_vent_in_heat:=FALSE;
				END_IF
			ELSE
				IF (Modbus.Vent_heat=1) THEN
					HW_vent_in_heat:=TRUE;
				(*	IF (Modbus.Vent_heat_level=TRUE) THEN
						HW_vent_in_heat_level:=TRUE;
					ELSE
						HW_vent_in_heat_level:=FALSE;
					END_IF
				*)
				END_IF
				IF (Modbus.Vent_heat=0) THEN
					HW_vent_in_heat:=FALSE;
				END_IF
			END_IF
		END_IF (*vent_relay_pressure*)
	END_IF (*vent_valve_opened*)
END_IF (*Vent*)
END_PROGRAM

(* POU VentPower, ST *)
PROGRAM VentPower
VAR
	Vent_power			: REAL:=30;	(* После перезагрузки ПЛК задаём начальную мощность приточного вента - условных 30%  *)
	Vent_power_out		: INT:=30;		(* После перезагрузки ПЛК задаём начальную мощность вытяжного вента - условных 30%  *)
	CO2_old				: REAL:=410;	(* После перезагрузки ПЛК задаём принудительно последнее значение CO2 = 410 (абсолютно свежий воздух) *)
	Period_vent_switch	: INT:=120; (* Период переключения режимов работы вентилятора по показаниям датчиков CO2, секунды*)
	Timer1				: TON;
	Timer1Q				: BOOL;
	count				: INT:=0;
	CO2_max			: REAL;
	tTimerValue			: TIME;

	Temp_low1			: REAL:=-19;
	Temp_low2			: REAL:=-23;



END_VAR
tTimerValue := DINT_TO_TIME(Period_vent_switch*1000);

IF (Modbus.Vent =TRUE OR Modbus.Vent_out=TRUE ) THEN

	Timer1(IN:=NOT Timer1Q , PT:=t#120s , Q=>Timer1Q , ET=> );
	IF timer1.q THEN
		CO2_max:=MAX(Internal.Kitchen_room_CO2, MAX (Internal.Bed_room_CO2, MAX (Internal.Child_big_room_CO2, Internal.Child_small_room_CO2)));
		IF (  (CO2_max >=  CO2_old-10 )  AND ( CO2_max >  INT_TO_REAL(Modbus.Target_CO2)*1.05 ) ) THEN
			Vent_power:=Vent_power+2;
		END_IF
		count:=count+1;
		IF (count = 5)	THEN
			IF (  CO2_max <=  INT_TO_REAL(Modbus.Target_CO2)*0.99) THEN
				Vent_power:=Vent_power-2;
			END_IF
			count:=1;
		END_IF

		IF (Vent_power>80) THEN
			Vent_power:=80;
		END_IF
		IF(Vent_power<20) THEN
			Vent_power:=20;
		END_IF

		IF (Vent_Power > 75  ) THEN

			IF (Internal.Kitchen_room_tempout  > Temp_low1 ) THEN
					Modbus.Vent_input_level:=200;									(* 200 м. куб в час при подаче напряжения на приточный вентилятор  220V *)
					HW_vent_in_trans_160_220:=FALSE;
					HW_vent_in_trans_LO_HI:=FALSE;
				ELSIF (Internal.Kitchen_room_tempout > Temp_low2 ) THEN
					Modbus.Vent_input_level:=150;							 (* 150 м. куб в час при подаче напряжения на приточный вентилятор  160V *)
					HW_vent_in_trans_160_220:=TRUE;
					HW_vent_in_trans_LO_HI:=FALSE;
				ELSE
					Modbus.Vent_input_level:=110; 								(* 110 м. куб в час при подаче напряжения на приточный вентилятор  130V *)
					HW_vent_in_trans_160_220:=FALSE;
					HW_vent_in_trans_LO_HI:=TRUE;
			END_IF

			IF (HW_kitchen_button_vent_out=FALSE) THEN					(* Если НЕ  работает кухонная надплитная вытяжка, то нужна тонкая регулировка вытяжного вента *)
				HW_vent_out_level:=REAL_TO_WORD(32767*60/100);			(* 200  м. куб в час при подаче x  DC напряжения на вытяжной вентилятор  *)
				Vent_power_out:=45;
			END_IF


		ELSIF (Vent_Power>50 ) THEN

			IF (Internal.Kitchen_room_tempout  > Temp_low1 ) THEN
					Modbus.Vent_input_level:=200;									(* 200 м. куб в час при подаче напряжения на приточный вентилятор  220V *)
					HW_vent_in_trans_160_220:=FALSE;
					HW_vent_in_trans_LO_HI:=FALSE;
				ELSIF (Internal.Kitchen_room_tempout > Temp_low2 ) THEN
					Modbus.Vent_input_level:=150;							 (* 150 м. куб в час при подаче напряжения на приточный вентилятор  160V *)
					HW_vent_in_trans_160_220:=TRUE;
					HW_vent_in_trans_LO_HI:=FALSE;
				ELSE
					Modbus.Vent_input_level:=110; 								(* 110 м. куб в час при подаче напряжения на приточный вентилятор  130V *)
					HW_vent_in_trans_160_220:=FALSE;
					HW_vent_in_trans_LO_HI:=TRUE;
			END_IF


			IF (HW_kitchen_button_vent_out=FALSE) THEN				(* Если НЕ  работает кухонная надплитная вытяжка, то нужна тонкая регулировка вытяжного вента *)
					HW_vent_out_level:=REAL_TO_WORD(32767*45/100); 		(* 180  м. куб в час при подаче x  DC напряжения на вытяжной вентилятор  *)
					Vent_power_out:=40;
			END_IF


		ELSIF (Vent_Power>35 AND Vent_Power<=50) THEN


			IF (Internal.Kitchen_room_tempout  > Temp_low2 ) THEN
					Modbus.Vent_input_level:=150;							 (* 150 м. куб в час при подаче напряжения на приточный вентилятор  160V *)
					HW_vent_in_trans_160_220:=TRUE;
					HW_vent_in_trans_LO_HI:=FALSE;
			ELSE
				Modbus.Vent_input_level:=110; 								(* 110 м. куб в час при подаче напряжения на приточный вентилятор  130V *)
				HW_vent_in_trans_160_220:=FALSE;
				HW_vent_in_trans_LO_HI:=TRUE;
			END_IF


			IF (HW_kitchen_button_vent_out=FALSE) THEN			(* Если НЕ  работает кухонная надплитная вытяжка, то нужна тонкая регулировка вытяжного вента *)
				HW_vent_out_level:=REAL_TO_WORD(32767*35/100);	(* 150  м. куб в час при подаче x  DC напряжения на вытяжной вентилятор  *)
				Vent_power_out:=35;
			END_IF

		ELSIF (Vent_Power>25 AND Vent_Power<=35) THEN

					Modbus.Vent_input_level:=110; (* 130V*)					 (* 110 м. куб в час при подаче напряжения на приточный вентилятор  130V *)
					HW_vent_in_trans_105_130:=FALSE;
					HW_vent_in_trans_LO_HI:=TRUE;
					IF (HW_kitchen_button_vent_out=FALSE) THEN			(* Если НЕ  работает кухонная надплитная вытяжка, то нужна тонкая регулировка вытяжного вента *)
						HW_vent_out_level:=REAL_TO_WORD(32767*25/100);	(* 110  м. куб в час при подаче x  DC напряжения на вытяжной вентилятор  *)
						Vent_power_out:=25;
					END_IF

			ELSE	(* Vent_Power > 80 *)

				Modbus.Vent_input_level:=80; (* 105V*)						 (* 80 м. куб в час при подаче напряжения на приточный вентилятор  105V *)
				HW_vent_in_trans_105_130:=TRUE;
				HW_vent_in_trans_LO_HI:=TRUE;
				IF (HW_kitchen_button_vent_out=FALSE) THEN				(* Если НЕ  работает кухонная надплитная вытяжка, то нужна тонкая регулировка вытяжного вента *)
					HW_vent_out_level:=REAL_TO_WORD(32767*20/100);		(* 80  м. куб в час при подаче x  DC напряжения на вытяжной вентилятор  *)
					Vent_power_out:=20;
				END_IF


			END_IF	(* Vent_Power > 80 *)
			CO2_old:=CO2_max;
			Modbus.Vent_output_level:=Vent_power_out;
	END_IF	(* Timer1 *)

ELSE	 (* Vent=TRUE*)

	Modbus.Vent_input_level:=0;
	IF (HW_kitchen_button_vent_out=FALSE) THEN
		HW_vent_out_level:=REAL_TO_WORD(32767*20/100);
	END_IF
	Modbus.Vent_output_level:=Vent_power_out;

END_IF   (* Vent=TRUE*)
END_PROGRAM

(* POU Counters, ST *)
PROGRAM Counters
VAR
	Trigger_bathroom_water_warm: F_TRIG;
	Trigger_bathroom_water_cold: F_TRIG;
	Trigger_kitchen_water_warm: F_TRIG;
	Trigger_kitchen_water_cold: F_TRIG;

END_VAR
Trigger_bathroom_water_warm(CLK :=HW_impulse_bathroom_water_warm);
Trigger_bathroom_water_cold(CLK :=HW_impulse_bathroom_water_cold);
Trigger_kitchen_water_warm(CLK :=HW_impulse_kitchen_water_warm);
Trigger_kitchen_water_cold(CLK :=HW_impulse_kitchen_water_cold);

IF (Trigger_bathroom_water_warm.Q) THEN
	Modbus.Bathroom_stat_warm_water:=Modbus.Bathroom_stat_warm_water+1;

END_IF

IF (Trigger_bathroom_water_cold.Q) THEN
	Modbus.Bathroom_stat_cold_water:=Modbus.Bathroom_stat_cold_water+1;
END_IF

IF (Trigger_kitchen_water_warm.Q) THEN
	Modbus.Kitchen_stat_warm_water:=Modbus.Kitchen_stat_warm_water+1;
END_IF

IF (Trigger_kitchen_water_cold.Q) THEN
	Modbus.Kitchen_stat_cold_water:=Modbus.Kitchen_stat_cold_water+1;
END_IF
END_PROGRAM

(* POU Fluid_bath, ST *)
PROGRAM Fluid_bath
VAR
	BUTTON3 	:	 R_TRIG;  (* Конпка №3 - переключение подачи воды в санузлах *)
END_VAR
Modbus.FLD_BATH:=HW_sensor_fld_van;
Modbus.FLD_PRC:=HW_sensor_fld_post;
Modbus.FLD_TLT:=HW_sensor_fld_tlt;


IF (Modbus.FLD_BATH=TRUE OR Modbus.FLD_PRC=TRUE OR Modbus.FLD_TLT=TRUE ) THEN
	HW_valve_water_bathroom:=FALSE;
	Modbus.FLD_valve_bathroom:=FALSE;
	Modbus.FLD_ALRM_BATH:=TRUE;
ELSE
	IF (Modbus.FLD_ALRM_BATH=FALSE) THEN
		HW_valve_water_bathroom:=TRUE;
		Modbus.FLD_valve_bathroom:=TRUE;
	ELSE
		HW_valve_water_bathroom:=FALSE;
		Modbus.FLD_valve_bathroom:=FALSE;
	END_IF
END_IF

BUTTON3 (CLK:=HW_IN03);

IF (     BUTTON3.Q ) THEN
	IF (Modbus.FLD_valve_bathroom=FALSE) THEN
		IF (Modbus.FLD_BATH=FALSE AND Modbus.FLD_PRC=FALSE AND Modbus.FLD_TLT=FALSE) THEN
			HW_valve_water_bathroom:=TRUE;
			Modbus.FLD_valve_bathroom:=TRUE;
			Modbus.FLD_ALRM_BATH:=FALSE;
		END_IF
	ELSE
		Modbus.FLD_ALRM_BATH:=TRUE;
		HW_valve_water_bathroom:=FALSE;
		Modbus.FLD_valve_bathroom:=FALSE;
	END_IF
END_IF
END_PROGRAM

(* POU Fluid_kitchen, ST *)
PROGRAM Fluid_kitchen
VAR
	BUTTON2 	:	 R_TRIG;  (* Конпка №2 - переключение подачи воды в кухне  *)
END_VAR
Modbus.FLD_KUH:=HW_sensor_fld_kitchen;



IF (Modbus.FLD_KUH=TRUE) THEN
	HW_valve_water_kitchen:=FALSE;
	Modbus.FLD_valve_kitchen:=FALSE;
	Modbus.FLD_ALRM_KITCHEN:=TRUE;
ELSE
	IF (Modbus.FLD_ALRM_KITCHEN=FALSE) THEN
		HW_valve_water_kitchen:=TRUE;
		Modbus.FLD_valve_kitchen:=TRUE;
	ELSE
		HW_valve_water_kitchen:=FALSE;
		Modbus.FLD_valve_kitchen:=FALSE;
	END_IF
END_IF

BUTTON2 (CLK:=HW_IN02);

IF ( BUTTON2.Q ) THEN
	IF (HW_valve_water_kitchen=FALSE) THEN
		IF (Modbus.FLD_KUH=FALSE) THEN
			HW_valve_water_kitchen:=TRUE;
			Modbus.FLD_valve_kitchen:=TRUE;
			Modbus.FLD_ALRM_KITCHEN:=FALSE;
		END_IF
	ELSE
		Modbus.FLD_ALRM_KITCHEN:=TRUE;
		HW_valve_water_kitchen:=FALSE;
		Modbus.FLD_valve_kitchen:=FALSE;
	END_IF
END_IF
END_PROGRAM

(* POU Light_hall, ST *)
PROGRAM Light_hall
VAR
	Timer1			: TOF;
	tTimerValue		: TIME;
	Period_light		: INT := 60;		(* Время работы светильника по датчику движения, секунды *)
END_VAR
tTimerValue := DINT_TO_TIME(Period_light*1000);
Timer1(IN:=(NOT HW_PIR_HALL OR NOT HW_PIR_door), PT:=tTimerValue);
(* HW_LIGHT_HALL:=Timer1.Q; *)
END_PROGRAM

(* POU FB_GET_CO2_MH_Z19B, ST *)
FUNCTION_BLOCK FB_GET_CO2_MH_Z19B
VAR_INPUT

END_VAR

VAR_OUTPUT
	co2				: REAL;
	done			: BOOL;
END_VAR

VAR
	SendBuffer		: ARRAY[0..8] OF BYTE :=16#FF,16#01,16#86,16#00,16#00,16#00,16#00,16#00,16#79;
	ReceiveBuffer	: ARRAY[0..13] OF BYTE;
	Clear			: ClearComBuffer;
	state			: INT:= 0;
	tmcheck			: TON;
	w_CO2		:	WORD;
(*
	Sensor_CO2_high	 			: BYTE;	
	Sensor_CO2_low 				: BYTE;
*)

END_VAR
tmcheck();

CASE state OF

0:
	done:=FALSE;
	Clear(Buffer := RxBufferCom1);
	SendDataCom1(pSendData:=ADR(SendBuffer),length:=9,TXbuffer:=TXBufferCom1,Busy=>,Error=>);
	tmCheck(in:=FALSE);
	tmCheck(in:=TRUE,pt:=t#2s);
	state:=1;

1: (*ответ*)

	ReceiveDataCom1(pPrefix:=,LenPrefix:=,pSuffix:=,LenSuffix:=,pReceiveData:=ADR(ReceiveBuffer),SizeReceiveData:=9,TImeOut:=t#1s,Reset:=,RXbuffer:=RxBufferCom1,DataReceived=>,busy=>,RxTimeout=>,LenReceiveData=>);

	IF ReceiveDataCom1.Error <> 0 THEN
		state:=9;
	END_IF

	IF ReceiveDataCom1.DataReceived THEN
		state:=2;
	ELSIF tmcheck.Q THEN
		 state:=9;
	END_IF;



2:(*расшифровка*)
	IF (ReceiveBuffer [0] = 16#FF AND ReceiveBuffer [1] = 16#86 ) THEN
(*		Sensor_CO2_high := ReceiveBuffer [2];
		Sensor_CO2_low := ReceiveBuffer [3];	*)
		MEMCPY(ADR(w_CO2),ADR(ReceiveBuffer[3]),1);
		MEMCPY(ADR(w_CO2)+1,ADR(ReceiveBuffer[2]),1);
		co2 := WORD_TO_REAL(w_CO2);

(*		IF (WORD_TO_REAL(w_CO2)<>0 AND WORD_TO_REAL(w_CO2)<5001) THEN
			co2 := WORD_TO_REAL(w_CO2);
			state:=10;
		ELSE
			state:=9;
		END_IF
*)

	ELSE
		state:=9;
	END_IF

9:
	co2:=0;
	done := TRUE;
	state:=0;
10:
	done := TRUE;
	state:=0;

END_CASE;
END_FUNCTION_BLOCK
